{attribute 'GeneratedUsingTerminal: AT2041-0250-0023'}
{attribute addProperty BoxType "AT2041-0250-0023"}
{attribute addProperty Id "A_0099_AT2040_5250_0018_AT2040_5250AT2040_33A3DF1B80"}
{attribute addProperty CRC "1371955884"}
{attribute addProperty Size "80"}
TYPE A_0045_AT2041_0250_0023_51C662AC EXTENDS AT2041_2EA6C9BF :
STRUCT
	{attribute addProperty Name "A_0099_AT2040_5250_0018_AT2040_5250"}
	{attribute addProperty PreviousPort "A_0045(AT2041-0250-0023) : B"}
	A_0099_AT2040_5250_0018_AT2040_5250 : AT2040_33A3DF1B;
END_STRUCT
END_TYPE

(* stored: Version 1.2.0.0, ProductVersion 3.1.4024.9
   DUT A_0045_AT2041_0250_0023_51C662AC: Id {a22e8f1e-8e58-4e14-b8f2-e10ddd67101a} *)
